Fanuc KAREL source: kd00042.KL

-- PROVISIONAL review KL for V1013-1; original PC SHA256 1ade363a620e334e250df25734aa7eed168926168e8232b3494516d54bcb0918
-- Incomplete behavior may be omitted. Consult companion uncertainty JSON. Do not deploy.
PROGRAM KD00042
%NOLOCKGROUP
VAR
  I : INTEGER
  J : INTEGER
  B : BOOLEAN
  R : REAL
  S : STRING[80]
-- UNRESOLVED_DECL N type=001100
BEGIN
  -- UNRESOLVED_PC offsets 5-12; opcodes 9D,23
  -- UNRESOLVED_PC offsets 17-21; opcodes 7F
END KD00042
